{attribute addProperty BoxType "EK1122-0000-0018"}
{attribute addProperty Id "A_0155_AX5191_0000_0212_AX5191_0000_0212AX5191_3FB01CDA28235.25Beckhoff_AX5xxxsub_EK1100EK1100_179A0949162A_0154_AX5118_0000_0011AX5118_47F5CC4725031.25A_0155_AX5125_0000_0011AX5125_47F5CC4725031.25A_0156_AX5201_0000_0011AX5201_D0280DF235444.25A_0157_AX5106_0000_0010AX5106_47F5CC4725031.25A_0158_AX5112_0000_0010AX5112_47F5CC4725031.25A_0159_AX5118_0000_0010AX5118_47F5CC4725031.25A_0160_AX5112_0000_0008AX5112_47F5CC4725031.25A_0161_AX5103_0000_0007AX5103_47F5CC4725031.25A_0162_AX5118_0000_0007AX5118_47F5CC4725031.25A_0163_AX5106_0000_0006AX5106_47F5CC4725031.25A_0164_AX5112_0000_0006AX5112_47F5CC4725031.25A_0165_AX5201_0000_0006AX5201_D0280DF235444.25A_0166_AX5101_0000_0005AX5101_47F5CC4725031.25A_0167_AX5103_0000_0005AX5103_47F5CC4725031.25A_0168_AX5203_0000_0005AX5203_D0280DF235444.25A_0169_AX5206_0000_0005AX5206_D0280DF235444.25A_0170_AX5101_0000_0004AX5101_47F5CC4725031.25A_0171_AX5103_0000_0004AX5103_47F5CC4725031.25A_0172_AX5206_0000_0004AX5206_D0280DF235444.25A_0173_AX5101_0000_0003AX5101_47F5CC4725031.25A_0174_AX5103_0000_0003AX5103_47F5CC4725031.25A_0175_AX5201_0000_0003AX5201_D0280DF235444.25A_0176_AX5203_0000_0003AX5203_D0280DF235444.25A_0177_AX5021_0000_0002AX5021_292ACD4718623.25A_0153_AX5206_0000_0200AX5206_7BA2318041852.25A_0152_AX5140_0000_0200AX5140_3FB01CDA28235.25A_0151_AX5118_0000_0200AX5118_3FB01CDA28235.25A_0150_AX5125_0000_0201AX5125_3FB01CDA28235.25A_0149_AX5101_0000_0202AX5101_3FB01CDA28235.25A_0148_AX5206_0000_0203AX5206_7BA2318041852.25A_0147_AX5172_0000_0203AX5172_3FB01CDA28235.25A_0146_AX5106_0000_0203AX5106_3FB01CDA28235.25A_0145_AX5206_0000_0210AX5206_7BA2318041852.25A_0144_AX5203_0000_0210AX5203_7BA2318041852.25A_0143_AX5193_0000_0210AX5193_3FB01CDA28235.25A_0142_AX5192_0000_0210AX5192_3FB01CDA28235.25A_0141_AX5191_0000_0210AX5191_3FB01CDA28235.25A_0140_AX5160_0000_0210AX5160_3FB01CDA28235.25A_0139_AX5140_0000_0210AX5140_3FB01CDA28235.25A_0138_AX5125_0000_0210AX5125_3FB01CDA28235.25A_0137_AX5112_0000_0210AX5112_3FB01CDA28235.25A_0136_AX5101_0000_0210AX5101_3FB01CDA28235.25A_0135_AX5206_0000_0212AX5206_7BA2318041852.25A_0134_AX5203_0000_0212AX5203_7BA2318041852.25A_0133_AX5172_0000_0212AX5172_3FB01CDA28235.25A_0132_AX5160_0000_0212AX5160_3FB01CDA28235.25A_0131_AX5125_0000_0212AX5125_3FB01CDA28235.25A_0130_AX5118_0000_0212AX5118_3FB01CDA28235.25A_0129_AX5106_0000_0212AX5106_3FB01CDA28235.25A_0128_AX5206_0000_0213AX5206_7BA2318041852.25A_0127_AX5101_0000_0213AX5101_3FB01CDA28235.25A_0081_AX5101_0000_0012AX5101_47F5CC4725031.25A_0082_AX5103_0000_0012AX5103_47F5CC4725031.25A_0083_AX5203_0000_0012AX5203_D0280DF235444.25A_0084_AX5101_0000_0011AX5101_47F5CC4725031.25A_0085_AX5203_0000_0011AX5203_D0280DF235444.25A_0086_AX5206_0000_0011AX5206_D0280DF235444.25A_0087_AX5101_0000_0010AX5101_47F5CC4725031.25A_0088_AX5103_0000_0010AX5103_47F5CC4725031.25A_0089_AX5125_0000_0010AX5125_47F5CC4725031.25A_0090_AX5201_0000_0010AX5201_D0280DF235444.25A_0091_AX5203_0000_0010AX5203_D0280DF235444.25A_0092_AX5206_0000_0010AX5206_D0280DF235444.25A_0093_AX5101_0000_0009AX5101_47F5CC4725031.25A_0094_AX5103_0000_0009AX5103_47F5CC4725031.25A_0095_AX5106_0000_0009AX5106_47F5CC4725031.25A_0096_AX5112_0000_0009AX5112_47F5CC4725031.25A_0097_AX5118_0000_0009AX5118_47F5CC4725031.25A_0098_AX5125_0000_0009AX5125_47F5CC4725031.25A_0099_AX5201_0000_0009AX5201_D0280DF235444.25A_0100_AX5203_0000_0009AX5203_D0280DF235444.25A_0101_AX5206_0000_0009AX5206_D0280DF235444.25A_0102_AX5101_0000_0008AX5101_47F5CC4725031.25A_0103_AX5103_0000_0008AX5103_47F5CC4725031.25A_0104_AX5106_0000_0008AX5106_47F5CC4725031.25A_0105_AX5118_0000_0008AX5118_47F5CC4725031.25A_0106_AX5125_0000_0008AX5125_47F5CC4725031.25A_0107_AX5201_0000_0008AX5201_D0280DF235444.25A_0108_AX5203_0000_0008AX5203_D0280DF235444.25A_0109_AX5206_0000_0008AX5206_D0280DF235444.25A_0110_AX5101_0000_0007AX5101_47F5CC4725031.25A_0111_AX5106_0000_0007AX5106_47F5CC4725031.25A_0112_AX5112_0000_0007AX5112_47F5CC4725031.25A_0113_AX5125_0000_0007AX5125_47F5CC4725031.25A_0114_AX5201_0000_0007AX5201_D0280DF235444.25A_0115_AX5203_0000_0007AX5203_D0280DF235444.25A_0116_AX5206_0000_0007AX5206_D0280DF235444.25A_0117_AX5101_0000_0006AX5101_47F5CC4725031.25A_0118_AX5103_0000_0006AX5103_47F5CC4725031.25A_0119_AX5203_0000_0006AX5203_D0280DF235444.25A_0120_AX5206_0000_0006AX5206_D0280DF235444.25A_0121_AX5106_0000_0005AX5106_47F5CC4725031.25A_0122_AX5201_0000_0005AX5201_D0280DF235444.25A_0123_AX5106_0000_0004AX5106_47F5CC4725031.25A_0124_AX5201_0000_0004AX5201_D0280DF235444.25A_0125_AX5203_0000_0004AX5203_D0280DF235444.25A_0126_AX5021_0000_0001AX5021_292ACD4718623.25A_0080_AX5203_0000_0200AX5203_7BA2318041852.25A_0079_AX5201_0000_0200AX5201_7BA2318041852.25A_0078_AX5125_0000_0200AX5125_3FB01CDA28235.25A_0077_AX5106_0000_0200AX5106_3FB01CDA28235.25A_0076_AX5101_0000_0200AX5101_3FB01CDA28235.25A_0075_AX5206_0000_0201AX5206_7BA2318041852.25A_0074_AX5203_0000_0201AX5203_7BA2318041852.25A_0073_AX5201_0000_0201AX5201_7BA2318041852.25A_0072_AX5172_0000_0201AX5172_3FB01CDA28235.25A_0071_AX5160_0000_0201AX5160_3FB01CDA28235.25A_0070_AX5140_0000_0201AX5140_3FB01CDA28235.25A_0069_AX5112_0000_0201AX5112_3FB01CDA28235.25A_0068_AX5103_0000_0201AX5103_3FB01CDA28235.25A_0067_AX5101_0000_0201AX5101_3FB01CDA28235.25A_0066_AX5206_0000_0202AX5206_7BA2318041852.25A_0065_AX5203_0000_0202AX5203_7BA2318041852.25A_0064_AX5201_0000_0202AX5201_7BA2318041852.25A_0063_AX5172_0000_0202AX5172_3FB01CDA28235.25A_0062_AX5160_0000_0202AX5160_3FB01CDA28235.25A_0061_AX5140_0000_0202AX5140_3FB01CDA28235.25A_0060_AX5125_0000_0202AX5125_3FB01CDA28235.25A_0059_AX5118_0000_0202AX5118_3FB01CDA28235.25A_0058_AX5112_0000_0202AX5112_3FB01CDA28235.25A_0057_AX5106_0000_0202AX5106_3FB01CDA28235.25A_0056_AX5103_0000_0202AX5103_3FB01CDA28235.25A_0055_AX5203_0000_0203AX5203_7BA2318041852.25A_0054_AX5201_0000_0203AX5201_7BA2318041852.25A_0053_AX5192_0000_0203AX5192_3FB01CDA28235.25A_0052_AX5191_0000_0203AX5191_3FB01CDA28235.25A_0051_AX5190_0000_0203AX5190_3FB01CDA28235.25A_0050_AX5160_0000_0203AX5160_3FB01CDA28235.25A_0049_AX5140_0000_0203AX5140_3FB01CDA28235.25A_0048_AX5125_0000_0203AX5125_3FB01CDA28235.25A_0047_AX5118_0000_0203AX5118_3FB01CDA28235.25A_0046_AX5112_0000_0203AX5112_3FB01CDA28235.25A_0045_AX5103_0000_0203AX5103_3FB01CDA28235.25A_0044_AX5101_0000_0203AX5101_3FB01CDA28235.25A_0043_AX5201_0000_0210AX5201_7BA2318041852.25A_0042_AX5190_0000_0210AX5190_3FB01CDA28235.25A_0041_AX5172_0000_0210AX5172_3FB01CDA28235.25A_0040_AX5118_0000_0210AX5118_3FB01CDA28235.25A_0039_AX5106_0000_0210AX5106_3FB01CDA28235.25A_0038_AX5201_0000_0212AX5201_7BA2318041852.25A_0037_AX5193_0000_0212AX5193_3FB01CDA28235.25A_0036_AX5192_0000_0212AX5192_3FB01CDA28235.25A_0035_AX5190_0000_0212AX5190_3FB01CDA28235.25A_0034_AX5140_0000_0212AX5140_3FB01CDA28235.25A_0033_AX5112_0000_0212AX5112_3FB01CDA28235.25A_0032_AX5103_0000_0212AX5103_3FB01CDA28235.25A_0031_AX5101_0000_0212AX5101_3FB01CDA28235.25A_0030_AX5203_0000_0213AX5203_7BA2318041852.25A_0029_AX5201_0000_0213AX5201_7BA2318041852.25A_0028_AX5193_0000_0213AX5193_3FB01CDA28235.25A_0027_AX5192_0000_0213AX5192_3FB01CDA28235.25A_0026_AX5191_0000_0213AX5191_3FB01CDA28235.25A_0025_AX5190_0000_0213AX5190_3FB01CDA28235.25A_0024_AX5172_0000_0213AX5172_3FB01CDA28235.25A_0023_AX5160_0000_0213AX5160_3FB01CDA28235.25A_0022_AX5140_0000_0213AX5140_3FB01CDA28235.25A_0021_AX5125_0000_0213AX5125_3FB01CDA28235.25A_0020_AX5118_0000_0213AX5118_3FB01CDA28235.25A_0019_AX5112_0000_0213AX5112_3FB01CDA28235.25A_0018_AX5106_0000_0213AX5106_3FB01CDA28235.25A_0017_AX5103_0000_0213AX5103_3FB01CDA28235.25A_0016_AX5206_0000_0214AX5206_7BA2318041852.25A_0015_AX5203_0000_0214AX5203_7BA2318041852.25A_0014_AX5201_0000_0214AX5201_7BA2318041852.25A_0013_AX5193_0000_0214AX5193_3FB01CDA28235.25A_0012_AX5192_0000_0214AX5192_3FB01CDA28235.25A_0011_AX5191_0000_0214AX5191_3FB01CDA28235.25A_0010_AX5190_0000_0214AX5190_3FB01CDA28235.25A_0009_AX5172_0000_0214AX5172_3FB01CDA28235.25A_0008_AX5160_0000_0214AX5160_3FB01CDA28235.25A_0007_AX5140_0000_0214AX5140_3FB01CDA28235.25A_0006_AX5125_0000_0214AX5125_3FB01CDA28235.25A_0005_AX5118_0000_0214AX5118_3FB01CDA28235.25A_0004_AX5112_0000_0214AX5112_3FB01CDA28235.25A_0003_AX5106_0000_0214AX5106_3FB01CDA28235.25A_0002_AX5103_0000_0214AX5103_3FB01CDA28235.25A_0001_AX5101_0000_0214AX5101_3FB01CDA28235.25A_0156_AX5103_0000_0210_AX5103_0000_0210AX5103_3FB01CDA28235.25A_0157_AX5193_0000_0203_AX5193_0000_0203AX5193_3FB01CDA28235.25A_0158_AX5106_0000_0201_AX5106_0000_0201AX5106_3FB01CDA28235.25A_0159_AX5118_0000_0201_AX5118_0000_0201AX5118_3FB01CDA28235.25A_0160_AX5103_0000_0200_AX5103_0000_0200AX5103_3FB01CDA28235.25A_0161_AX5112_0000_0200_AX5112_0000_0200AX5112_3FB01CDA28235.25A_0162_AX5106_0000_0012_AX5106_0000_0012AX5106_47F5CC4725031.25A_0163_AX5112_0000_0012_AX5112_0000_0012AX5112_47F5CC4725031.25A_0164_AX5118_0000_0012_AX5118_0000_0012AX5118_47F5CC4725031.25A_0165_AX5125_0000_0012_AX5125_0000_0012AX5125_47F5CC4725031.25A_0166_AX5201_0000_0012_AX5201_0000_0012AX5201_D0280DF235444.25A_0167_AX5206_0000_0012_AX5206_0000_0012AX5206_D0280DF235444.25A_0168_AX5103_0000_0011AX5103_47F5CC4725031.25A_0169_AX5106_0000_0011_AX5106_0000_0011AX5106_47F5CC4725031.25A_0170_AX5112_0000_0011_AX5112_0000_0011AX5112_47F5CC4725031.25A_0171_AX5106_0000_0003_AX5106_0000_0003AX5106_47F5CC4725031.25A_0172_AX5206_0000_0003_AX5206_0000_0003AX5206_D0280DF235444.25"}
{attribute addProperty CRC "1593486659"}
{attribute addProperty SizeInBites "58670"}
{attribute addProperty SizeInBytes "7333.75"}
TYPE Beckhoff_AX5xxxEK1122_5EFAAD43 EXTENDS EK1122_179A0949 :
STRUCT
	{attribute addProperty Name "A_0155_AX5191_0000_0212_AX5191_0000_0212"}
	A_0155_AX5191_0000_0212_AX5191_0000_0212 : AX5191_3FB01CDA;
	{attribute addProperty Name "Beckhoff_AX5xxxsub_EK1100"}
	Beckhoff_AX5xxxsub_EK1100 : EK1100_179A0949;
	{attribute addProperty Name "A_0154_AX5118_0000_0011"}
	A_0154_AX5118_0000_0011 : AX5118_47F5CC47;
	{attribute addProperty Name "A_0155_AX5125_0000_0011"}
	A_0155_AX5125_0000_0011 : AX5125_47F5CC47;
	{attribute addProperty Name "A_0156_AX5201_0000_0011"}
	A_0156_AX5201_0000_0011 : AX5201_D0280DF2;
	{attribute addProperty Name "A_0157_AX5106_0000_0010"}
	A_0157_AX5106_0000_0010 : AX5106_47F5CC47;
	{attribute addProperty Name "A_0158_AX5112_0000_0010"}
	A_0158_AX5112_0000_0010 : AX5112_47F5CC47;
	{attribute addProperty Name "A_0159_AX5118_0000_0010"}
	A_0159_AX5118_0000_0010 : AX5118_47F5CC47;
	{attribute addProperty Name "A_0160_AX5112_0000_0008"}
	A_0160_AX5112_0000_0008 : AX5112_47F5CC47;
	{attribute addProperty Name "A_0161_AX5103_0000_0007"}
	A_0161_AX5103_0000_0007 : AX5103_47F5CC47;
	{attribute addProperty Name "A_0162_AX5118_0000_0007"}
	A_0162_AX5118_0000_0007 : AX5118_47F5CC47;
	{attribute addProperty Name "A_0163_AX5106_0000_0006"}
	A_0163_AX5106_0000_0006 : AX5106_47F5CC47;
	{attribute addProperty Name "A_0164_AX5112_0000_0006"}
	A_0164_AX5112_0000_0006 : AX5112_47F5CC47;
	{attribute addProperty Name "A_0165_AX5201_0000_0006"}
	A_0165_AX5201_0000_0006 : AX5201_D0280DF2;
	{attribute addProperty Name "A_0166_AX5101_0000_0005"}
	A_0166_AX5101_0000_0005 : AX5101_47F5CC47;
	{attribute addProperty Name "A_0167_AX5103_0000_0005"}
	A_0167_AX5103_0000_0005 : AX5103_47F5CC47;
	{attribute addProperty Name "A_0168_AX5203_0000_0005"}
	A_0168_AX5203_0000_0005 : AX5203_D0280DF2;
	{attribute addProperty Name "A_0169_AX5206_0000_0005"}
	A_0169_AX5206_0000_0005 : AX5206_D0280DF2;
	{attribute addProperty Name "A_0170_AX5101_0000_0004"}
	A_0170_AX5101_0000_0004 : AX5101_47F5CC47;
	{attribute addProperty Name "A_0171_AX5103_0000_0004"}
	A_0171_AX5103_0000_0004 : AX5103_47F5CC47;
	{attribute addProperty Name "A_0172_AX5206_0000_0004"}
	A_0172_AX5206_0000_0004 : AX5206_D0280DF2;
	{attribute addProperty Name "A_0173_AX5101_0000_0003"}
	A_0173_AX5101_0000_0003 : AX5101_47F5CC47;
	{attribute addProperty Name "A_0174_AX5103_0000_0003"}
	A_0174_AX5103_0000_0003 : AX5103_47F5CC47;
	{attribute addProperty Name "A_0175_AX5201_0000_0003"}
	A_0175_AX5201_0000_0003 : AX5201_D0280DF2;
	{attribute addProperty Name "A_0176_AX5203_0000_0003"}
	A_0176_AX5203_0000_0003 : AX5203_D0280DF2;
	{attribute addProperty Name "A_0177_AX5021_0000_0002"}
	A_0177_AX5021_0000_0002 : AX5021_292ACD47;
	{attribute addProperty Name "A_0153_AX5206_0000_0200"}
	A_0153_AX5206_0000_0200 : AX5206_7BA23180;
	{attribute addProperty Name "A_0152_AX5140_0000_0200"}
	A_0152_AX5140_0000_0200 : AX5140_3FB01CDA;
	{attribute addProperty Name "A_0151_AX5118_0000_0200"}
	A_0151_AX5118_0000_0200 : AX5118_3FB01CDA;
	{attribute addProperty Name "A_0150_AX5125_0000_0201"}
	A_0150_AX5125_0000_0201 : AX5125_3FB01CDA;
	{attribute addProperty Name "A_0149_AX5101_0000_0202"}
	A_0149_AX5101_0000_0202 : AX5101_3FB01CDA;
	{attribute addProperty Name "A_0148_AX5206_0000_0203"}
	A_0148_AX5206_0000_0203 : AX5206_7BA23180;
	{attribute addProperty Name "A_0147_AX5172_0000_0203"}
	A_0147_AX5172_0000_0203 : AX5172_3FB01CDA;
	{attribute addProperty Name "A_0146_AX5106_0000_0203"}
	A_0146_AX5106_0000_0203 : AX5106_3FB01CDA;
	{attribute addProperty Name "A_0145_AX5206_0000_0210"}
	A_0145_AX5206_0000_0210 : AX5206_7BA23180;
	{attribute addProperty Name "A_0144_AX5203_0000_0210"}
	A_0144_AX5203_0000_0210 : AX5203_7BA23180;
	{attribute addProperty Name "A_0143_AX5193_0000_0210"}
	A_0143_AX5193_0000_0210 : AX5193_3FB01CDA;
	{attribute addProperty Name "A_0142_AX5192_0000_0210"}
	A_0142_AX5192_0000_0210 : AX5192_3FB01CDA;
	{attribute addProperty Name "A_0141_AX5191_0000_0210"}
	A_0141_AX5191_0000_0210 : AX5191_3FB01CDA;
	{attribute addProperty Name "A_0140_AX5160_0000_0210"}
	A_0140_AX5160_0000_0210 : AX5160_3FB01CDA;
	{attribute addProperty Name "A_0139_AX5140_0000_0210"}
	A_0139_AX5140_0000_0210 : AX5140_3FB01CDA;
	{attribute addProperty Name "A_0138_AX5125_0000_0210"}
	A_0138_AX5125_0000_0210 : AX5125_3FB01CDA;
	{attribute addProperty Name "A_0137_AX5112_0000_0210"}
	A_0137_AX5112_0000_0210 : AX5112_3FB01CDA;
	{attribute addProperty Name "A_0136_AX5101_0000_0210"}
	A_0136_AX5101_0000_0210 : AX5101_3FB01CDA;
	{attribute addProperty Name "A_0135_AX5206_0000_0212"}
	A_0135_AX5206_0000_0212 : AX5206_7BA23180;
	{attribute addProperty Name "A_0134_AX5203_0000_0212"}
	A_0134_AX5203_0000_0212 : AX5203_7BA23180;
	{attribute addProperty Name "A_0133_AX5172_0000_0212"}
	A_0133_AX5172_0000_0212 : AX5172_3FB01CDA;
	{attribute addProperty Name "A_0132_AX5160_0000_0212"}
	A_0132_AX5160_0000_0212 : AX5160_3FB01CDA;
	{attribute addProperty Name "A_0131_AX5125_0000_0212"}
	A_0131_AX5125_0000_0212 : AX5125_3FB01CDA;
	{attribute addProperty Name "A_0130_AX5118_0000_0212"}
	A_0130_AX5118_0000_0212 : AX5118_3FB01CDA;
	{attribute addProperty Name "A_0129_AX5106_0000_0212"}
	A_0129_AX5106_0000_0212 : AX5106_3FB01CDA;
	{attribute addProperty Name "A_0128_AX5206_0000_0213"}
	A_0128_AX5206_0000_0213 : AX5206_7BA23180;
	{attribute addProperty Name "A_0127_AX5101_0000_0213"}
	A_0127_AX5101_0000_0213 : AX5101_3FB01CDA;
	{attribute addProperty Name "A_0081_AX5101_0000_0012"}
	A_0081_AX5101_0000_0012 : AX5101_47F5CC47;
	{attribute addProperty Name "A_0082_AX5103_0000_0012"}
	A_0082_AX5103_0000_0012 : AX5103_47F5CC47;
	{attribute addProperty Name "A_0083_AX5203_0000_0012"}
	A_0083_AX5203_0000_0012 : AX5203_D0280DF2;
	{attribute addProperty Name "A_0084_AX5101_0000_0011"}
	A_0084_AX5101_0000_0011 : AX5101_47F5CC47;
	{attribute addProperty Name "A_0085_AX5203_0000_0011"}
	A_0085_AX5203_0000_0011 : AX5203_D0280DF2;
	{attribute addProperty Name "A_0086_AX5206_0000_0011"}
	A_0086_AX5206_0000_0011 : AX5206_D0280DF2;
	{attribute addProperty Name "A_0087_AX5101_0000_0010"}
	A_0087_AX5101_0000_0010 : AX5101_47F5CC47;
	{attribute addProperty Name "A_0088_AX5103_0000_0010"}
	A_0088_AX5103_0000_0010 : AX5103_47F5CC47;
	{attribute addProperty Name "A_0089_AX5125_0000_0010"}
	A_0089_AX5125_0000_0010 : AX5125_47F5CC47;
	{attribute addProperty Name "A_0090_AX5201_0000_0010"}
	A_0090_AX5201_0000_0010 : AX5201_D0280DF2;
	{attribute addProperty Name "A_0091_AX5203_0000_0010"}
	A_0091_AX5203_0000_0010 : AX5203_D0280DF2;
	{attribute addProperty Name "A_0092_AX5206_0000_0010"}
	A_0092_AX5206_0000_0010 : AX5206_D0280DF2;
	{attribute addProperty Name "A_0093_AX5101_0000_0009"}
	A_0093_AX5101_0000_0009 : AX5101_47F5CC47;
	{attribute addProperty Name "A_0094_AX5103_0000_0009"}
	A_0094_AX5103_0000_0009 : AX5103_47F5CC47;
	{attribute addProperty Name "A_0095_AX5106_0000_0009"}
	A_0095_AX5106_0000_0009 : AX5106_47F5CC47;
	{attribute addProperty Name "A_0096_AX5112_0000_0009"}
	A_0096_AX5112_0000_0009 : AX5112_47F5CC47;
	{attribute addProperty Name "A_0097_AX5118_0000_0009"}
	A_0097_AX5118_0000_0009 : AX5118_47F5CC47;
	{attribute addProperty Name "A_0098_AX5125_0000_0009"}
	A_0098_AX5125_0000_0009 : AX5125_47F5CC47;
	{attribute addProperty Name "A_0099_AX5201_0000_0009"}
	A_0099_AX5201_0000_0009 : AX5201_D0280DF2;
	{attribute addProperty Name "A_0100_AX5203_0000_0009"}
	A_0100_AX5203_0000_0009 : AX5203_D0280DF2;
	{attribute addProperty Name "A_0101_AX5206_0000_0009"}
	A_0101_AX5206_0000_0009 : AX5206_D0280DF2;
	{attribute addProperty Name "A_0102_AX5101_0000_0008"}
	A_0102_AX5101_0000_0008 : AX5101_47F5CC47;
	{attribute addProperty Name "A_0103_AX5103_0000_0008"}
	A_0103_AX5103_0000_0008 : AX5103_47F5CC47;
	{attribute addProperty Name "A_0104_AX5106_0000_0008"}
	A_0104_AX5106_0000_0008 : AX5106_47F5CC47;
	{attribute addProperty Name "A_0105_AX5118_0000_0008"}
	A_0105_AX5118_0000_0008 : AX5118_47F5CC47;
	{attribute addProperty Name "A_0106_AX5125_0000_0008"}
	A_0106_AX5125_0000_0008 : AX5125_47F5CC47;
	{attribute addProperty Name "A_0107_AX5201_0000_0008"}
	A_0107_AX5201_0000_0008 : AX5201_D0280DF2;
	{attribute addProperty Name "A_0108_AX5203_0000_0008"}
	A_0108_AX5203_0000_0008 : AX5203_D0280DF2;
	{attribute addProperty Name "A_0109_AX5206_0000_0008"}
	A_0109_AX5206_0000_0008 : AX5206_D0280DF2;
	{attribute addProperty Name "A_0110_AX5101_0000_0007"}
	A_0110_AX5101_0000_0007 : AX5101_47F5CC47;
	{attribute addProperty Name "A_0111_AX5106_0000_0007"}
	A_0111_AX5106_0000_0007 : AX5106_47F5CC47;
	{attribute addProperty Name "A_0112_AX5112_0000_0007"}
	A_0112_AX5112_0000_0007 : AX5112_47F5CC47;
	{attribute addProperty Name "A_0113_AX5125_0000_0007"}
	A_0113_AX5125_0000_0007 : AX5125_47F5CC47;
	{attribute addProperty Name "A_0114_AX5201_0000_0007"}
	A_0114_AX5201_0000_0007 : AX5201_D0280DF2;
	{attribute addProperty Name "A_0115_AX5203_0000_0007"}
	A_0115_AX5203_0000_0007 : AX5203_D0280DF2;
	{attribute addProperty Name "A_0116_AX5206_0000_0007"}
	A_0116_AX5206_0000_0007 : AX5206_D0280DF2;
	{attribute addProperty Name "A_0117_AX5101_0000_0006"}
	A_0117_AX5101_0000_0006 : AX5101_47F5CC47;
	{attribute addProperty Name "A_0118_AX5103_0000_0006"}
	A_0118_AX5103_0000_0006 : AX5103_47F5CC47;
	{attribute addProperty Name "A_0119_AX5203_0000_0006"}
	A_0119_AX5203_0000_0006 : AX5203_D0280DF2;
	{attribute addProperty Name "A_0120_AX5206_0000_0006"}
	A_0120_AX5206_0000_0006 : AX5206_D0280DF2;
	{attribute addProperty Name "A_0121_AX5106_0000_0005"}
	A_0121_AX5106_0000_0005 : AX5106_47F5CC47;
	{attribute addProperty Name "A_0122_AX5201_0000_0005"}
	A_0122_AX5201_0000_0005 : AX5201_D0280DF2;
	{attribute addProperty Name "A_0123_AX5106_0000_0004"}
	A_0123_AX5106_0000_0004 : AX5106_47F5CC47;
	{attribute addProperty Name "A_0124_AX5201_0000_0004"}
	A_0124_AX5201_0000_0004 : AX5201_D0280DF2;
	{attribute addProperty Name "A_0125_AX5203_0000_0004"}
	A_0125_AX5203_0000_0004 : AX5203_D0280DF2;
	{attribute addProperty Name "A_0126_AX5021_0000_0001"}
	A_0126_AX5021_0000_0001 : AX5021_292ACD47;
	{attribute addProperty Name "A_0080_AX5203_0000_0200"}
	A_0080_AX5203_0000_0200 : AX5203_7BA23180;
	{attribute addProperty Name "A_0079_AX5201_0000_0200"}
	A_0079_AX5201_0000_0200 : AX5201_7BA23180;
	{attribute addProperty Name "A_0078_AX5125_0000_0200"}
	A_0078_AX5125_0000_0200 : AX5125_3FB01CDA;
	{attribute addProperty Name "A_0077_AX5106_0000_0200"}
	A_0077_AX5106_0000_0200 : AX5106_3FB01CDA;
	{attribute addProperty Name "A_0076_AX5101_0000_0200"}
	A_0076_AX5101_0000_0200 : AX5101_3FB01CDA;
	{attribute addProperty Name "A_0075_AX5206_0000_0201"}
	A_0075_AX5206_0000_0201 : AX5206_7BA23180;
	{attribute addProperty Name "A_0074_AX5203_0000_0201"}
	A_0074_AX5203_0000_0201 : AX5203_7BA23180;
	{attribute addProperty Name "A_0073_AX5201_0000_0201"}
	A_0073_AX5201_0000_0201 : AX5201_7BA23180;
	{attribute addProperty Name "A_0072_AX5172_0000_0201"}
	A_0072_AX5172_0000_0201 : AX5172_3FB01CDA;
	{attribute addProperty Name "A_0071_AX5160_0000_0201"}
	A_0071_AX5160_0000_0201 : AX5160_3FB01CDA;
	{attribute addProperty Name "A_0070_AX5140_0000_0201"}
	A_0070_AX5140_0000_0201 : AX5140_3FB01CDA;
	{attribute addProperty Name "A_0069_AX5112_0000_0201"}
	A_0069_AX5112_0000_0201 : AX5112_3FB01CDA;
	{attribute addProperty Name "A_0068_AX5103_0000_0201"}
	A_0068_AX5103_0000_0201 : AX5103_3FB01CDA;
	{attribute addProperty Name "A_0067_AX5101_0000_0201"}
	A_0067_AX5101_0000_0201 : AX5101_3FB01CDA;
	{attribute addProperty Name "A_0066_AX5206_0000_0202"}
	A_0066_AX5206_0000_0202 : AX5206_7BA23180;
	{attribute addProperty Name "A_0065_AX5203_0000_0202"}
	A_0065_AX5203_0000_0202 : AX5203_7BA23180;
	{attribute addProperty Name "A_0064_AX5201_0000_0202"}
	A_0064_AX5201_0000_0202 : AX5201_7BA23180;
	{attribute addProperty Name "A_0063_AX5172_0000_0202"}
	A_0063_AX5172_0000_0202 : AX5172_3FB01CDA;
	{attribute addProperty Name "A_0062_AX5160_0000_0202"}
	A_0062_AX5160_0000_0202 : AX5160_3FB01CDA;
	{attribute addProperty Name "A_0061_AX5140_0000_0202"}
	A_0061_AX5140_0000_0202 : AX5140_3FB01CDA;
	{attribute addProperty Name "A_0060_AX5125_0000_0202"}
	A_0060_AX5125_0000_0202 : AX5125_3FB01CDA;
	{attribute addProperty Name "A_0059_AX5118_0000_0202"}
	A_0059_AX5118_0000_0202 : AX5118_3FB01CDA;
	{attribute addProperty Name "A_0058_AX5112_0000_0202"}
	A_0058_AX5112_0000_0202 : AX5112_3FB01CDA;
	{attribute addProperty Name "A_0057_AX5106_0000_0202"}
	A_0057_AX5106_0000_0202 : AX5106_3FB01CDA;
	{attribute addProperty Name "A_0056_AX5103_0000_0202"}
	A_0056_AX5103_0000_0202 : AX5103_3FB01CDA;
	{attribute addProperty Name "A_0055_AX5203_0000_0203"}
	A_0055_AX5203_0000_0203 : AX5203_7BA23180;
	{attribute addProperty Name "A_0054_AX5201_0000_0203"}
	A_0054_AX5201_0000_0203 : AX5201_7BA23180;
	{attribute addProperty Name "A_0053_AX5192_0000_0203"}
	A_0053_AX5192_0000_0203 : AX5192_3FB01CDA;
	{attribute addProperty Name "A_0052_AX5191_0000_0203"}
	A_0052_AX5191_0000_0203 : AX5191_3FB01CDA;
	{attribute addProperty Name "A_0051_AX5190_0000_0203"}
	A_0051_AX5190_0000_0203 : AX5190_3FB01CDA;
	{attribute addProperty Name "A_0050_AX5160_0000_0203"}
	A_0050_AX5160_0000_0203 : AX5160_3FB01CDA;
	{attribute addProperty Name "A_0049_AX5140_0000_0203"}
	A_0049_AX5140_0000_0203 : AX5140_3FB01CDA;
	{attribute addProperty Name "A_0048_AX5125_0000_0203"}
	A_0048_AX5125_0000_0203 : AX5125_3FB01CDA;
	{attribute addProperty Name "A_0047_AX5118_0000_0203"}
	A_0047_AX5118_0000_0203 : AX5118_3FB01CDA;
	{attribute addProperty Name "A_0046_AX5112_0000_0203"}
	A_0046_AX5112_0000_0203 : AX5112_3FB01CDA;
	{attribute addProperty Name "A_0045_AX5103_0000_0203"}
	A_0045_AX5103_0000_0203 : AX5103_3FB01CDA;
	{attribute addProperty Name "A_0044_AX5101_0000_0203"}
	A_0044_AX5101_0000_0203 : AX5101_3FB01CDA;
	{attribute addProperty Name "A_0043_AX5201_0000_0210"}
	A_0043_AX5201_0000_0210 : AX5201_7BA23180;
	{attribute addProperty Name "A_0042_AX5190_0000_0210"}
	A_0042_AX5190_0000_0210 : AX5190_3FB01CDA;
	{attribute addProperty Name "A_0041_AX5172_0000_0210"}
	A_0041_AX5172_0000_0210 : AX5172_3FB01CDA;
	{attribute addProperty Name "A_0040_AX5118_0000_0210"}
	A_0040_AX5118_0000_0210 : AX5118_3FB01CDA;
	{attribute addProperty Name "A_0039_AX5106_0000_0210"}
	A_0039_AX5106_0000_0210 : AX5106_3FB01CDA;
	{attribute addProperty Name "A_0038_AX5201_0000_0212"}
	A_0038_AX5201_0000_0212 : AX5201_7BA23180;
	{attribute addProperty Name "A_0037_AX5193_0000_0212"}
	A_0037_AX5193_0000_0212 : AX5193_3FB01CDA;
	{attribute addProperty Name "A_0036_AX5192_0000_0212"}
	A_0036_AX5192_0000_0212 : AX5192_3FB01CDA;
	{attribute addProperty Name "A_0035_AX5190_0000_0212"}
	A_0035_AX5190_0000_0212 : AX5190_3FB01CDA;
	{attribute addProperty Name "A_0034_AX5140_0000_0212"}
	A_0034_AX5140_0000_0212 : AX5140_3FB01CDA;
	{attribute addProperty Name "A_0033_AX5112_0000_0212"}
	A_0033_AX5112_0000_0212 : AX5112_3FB01CDA;
	{attribute addProperty Name "A_0032_AX5103_0000_0212"}
	A_0032_AX5103_0000_0212 : AX5103_3FB01CDA;
	{attribute addProperty Name "A_0031_AX5101_0000_0212"}
	A_0031_AX5101_0000_0212 : AX5101_3FB01CDA;
	{attribute addProperty Name "A_0030_AX5203_0000_0213"}
	A_0030_AX5203_0000_0213 : AX5203_7BA23180;
	{attribute addProperty Name "A_0029_AX5201_0000_0213"}
	A_0029_AX5201_0000_0213 : AX5201_7BA23180;
	{attribute addProperty Name "A_0028_AX5193_0000_0213"}
	A_0028_AX5193_0000_0213 : AX5193_3FB01CDA;
	{attribute addProperty Name "A_0027_AX5192_0000_0213"}
	A_0027_AX5192_0000_0213 : AX5192_3FB01CDA;
	{attribute addProperty Name "A_0026_AX5191_0000_0213"}
	A_0026_AX5191_0000_0213 : AX5191_3FB01CDA;
	{attribute addProperty Name "A_0025_AX5190_0000_0213"}
	A_0025_AX5190_0000_0213 : AX5190_3FB01CDA;
	{attribute addProperty Name "A_0024_AX5172_0000_0213"}
	A_0024_AX5172_0000_0213 : AX5172_3FB01CDA;
	{attribute addProperty Name "A_0023_AX5160_0000_0213"}
	A_0023_AX5160_0000_0213 : AX5160_3FB01CDA;
	{attribute addProperty Name "A_0022_AX5140_0000_0213"}
	A_0022_AX5140_0000_0213 : AX5140_3FB01CDA;
	{attribute addProperty Name "A_0021_AX5125_0000_0213"}
	A_0021_AX5125_0000_0213 : AX5125_3FB01CDA;
	{attribute addProperty Name "A_0020_AX5118_0000_0213"}
	A_0020_AX5118_0000_0213 : AX5118_3FB01CDA;
	{attribute addProperty Name "A_0019_AX5112_0000_0213"}
	A_0019_AX5112_0000_0213 : AX5112_3FB01CDA;
	{attribute addProperty Name "A_0018_AX5106_0000_0213"}
	A_0018_AX5106_0000_0213 : AX5106_3FB01CDA;
	{attribute addProperty Name "A_0017_AX5103_0000_0213"}
	A_0017_AX5103_0000_0213 : AX5103_3FB01CDA;
	{attribute addProperty Name "A_0016_AX5206_0000_0214"}
	A_0016_AX5206_0000_0214 : AX5206_7BA23180;
	{attribute addProperty Name "A_0015_AX5203_0000_0214"}
	A_0015_AX5203_0000_0214 : AX5203_7BA23180;
	{attribute addProperty Name "A_0014_AX5201_0000_0214"}
	A_0014_AX5201_0000_0214 : AX5201_7BA23180;
	{attribute addProperty Name "A_0013_AX5193_0000_0214"}
	A_0013_AX5193_0000_0214 : AX5193_3FB01CDA;
	{attribute addProperty Name "A_0012_AX5192_0000_0214"}
	A_0012_AX5192_0000_0214 : AX5192_3FB01CDA;
	{attribute addProperty Name "A_0011_AX5191_0000_0214"}
	A_0011_AX5191_0000_0214 : AX5191_3FB01CDA;
	{attribute addProperty Name "A_0010_AX5190_0000_0214"}
	A_0010_AX5190_0000_0214 : AX5190_3FB01CDA;
	{attribute addProperty Name "A_0009_AX5172_0000_0214"}
	A_0009_AX5172_0000_0214 : AX5172_3FB01CDA;
	{attribute addProperty Name "A_0008_AX5160_0000_0214"}
	A_0008_AX5160_0000_0214 : AX5160_3FB01CDA;
	{attribute addProperty Name "A_0007_AX5140_0000_0214"}
	A_0007_AX5140_0000_0214 : AX5140_3FB01CDA;
	{attribute addProperty Name "A_0006_AX5125_0000_0214"}
	A_0006_AX5125_0000_0214 : AX5125_3FB01CDA;
	{attribute addProperty Name "A_0005_AX5118_0000_0214"}
	A_0005_AX5118_0000_0214 : AX5118_3FB01CDA;
	{attribute addProperty Name "A_0004_AX5112_0000_0214"}
	A_0004_AX5112_0000_0214 : AX5112_3FB01CDA;
	{attribute addProperty Name "A_0003_AX5106_0000_0214"}
	A_0003_AX5106_0000_0214 : AX5106_3FB01CDA;
	{attribute addProperty Name "A_0002_AX5103_0000_0214"}
	A_0002_AX5103_0000_0214 : AX5103_3FB01CDA;
	{attribute addProperty Name "A_0001_AX5101_0000_0214"}
	A_0001_AX5101_0000_0214 : AX5101_3FB01CDA;
	{attribute addProperty Name "A_0156_AX5103_0000_0210_AX5103_0000_0210"}
	A_0156_AX5103_0000_0210_AX5103_0000_0210 : AX5103_3FB01CDA;
	{attribute addProperty Name "A_0157_AX5193_0000_0203_AX5193_0000_0203"}
	A_0157_AX5193_0000_0203_AX5193_0000_0203 : AX5193_3FB01CDA;
	{attribute addProperty Name "A_0158_AX5106_0000_0201_AX5106_0000_0201"}
	A_0158_AX5106_0000_0201_AX5106_0000_0201 : AX5106_3FB01CDA;
	{attribute addProperty Name "A_0159_AX5118_0000_0201_AX5118_0000_0201"}
	A_0159_AX5118_0000_0201_AX5118_0000_0201 : AX5118_3FB01CDA;
	{attribute addProperty Name "A_0160_AX5103_0000_0200_AX5103_0000_0200"}
	A_0160_AX5103_0000_0200_AX5103_0000_0200 : AX5103_3FB01CDA;
	{attribute addProperty Name "A_0161_AX5112_0000_0200_AX5112_0000_0200"}
	A_0161_AX5112_0000_0200_AX5112_0000_0200 : AX5112_3FB01CDA;
	{attribute addProperty Name "A_0162_AX5106_0000_0012_AX5106_0000_0012"}
	A_0162_AX5106_0000_0012_AX5106_0000_0012 : AX5106_47F5CC47;
	{attribute addProperty Name "A_0163_AX5112_0000_0012_AX5112_0000_0012"}
	A_0163_AX5112_0000_0012_AX5112_0000_0012 : AX5112_47F5CC47;
	{attribute addProperty Name "A_0164_AX5118_0000_0012_AX5118_0000_0012"}
	A_0164_AX5118_0000_0012_AX5118_0000_0012 : AX5118_47F5CC47;
	{attribute addProperty Name "A_0165_AX5125_0000_0012_AX5125_0000_0012"}
	A_0165_AX5125_0000_0012_AX5125_0000_0012 : AX5125_47F5CC47;
	{attribute addProperty Name "A_0166_AX5201_0000_0012_AX5201_0000_0012"}
	A_0166_AX5201_0000_0012_AX5201_0000_0012 : AX5201_D0280DF2;
	{attribute addProperty Name "A_0167_AX5206_0000_0012_AX5206_0000_0012"}
	A_0167_AX5206_0000_0012_AX5206_0000_0012 : AX5206_D0280DF2;
	{attribute addProperty Name "A_0168_AX5103_0000_0011"}
	A_0168_AX5103_0000_0011 : AX5103_47F5CC47;
	{attribute addProperty Name "A_0169_AX5106_0000_0011_AX5106_0000_0011"}
	A_0169_AX5106_0000_0011_AX5106_0000_0011 : AX5106_47F5CC47;
	{attribute addProperty Name "A_0170_AX5112_0000_0011_AX5112_0000_0011"}
	A_0170_AX5112_0000_0011_AX5112_0000_0011 : AX5112_47F5CC47;
	{attribute addProperty Name "A_0171_AX5106_0000_0003_AX5106_0000_0003"}
	A_0171_AX5106_0000_0003_AX5106_0000_0003 : AX5106_47F5CC47;
	{attribute addProperty Name "A_0172_AX5206_0000_0003_AX5206_0000_0003"}
	A_0172_AX5206_0000_0003_AX5206_0000_0003 : AX5206_D0280DF2;
END_STRUCT
END_TYPE

(* stored: Version 1.2.0.0, ProductVersion 3.1.4024.9
   DUT Beckhoff_AX5xxxEK1122_5EFAAD43: Id {e8651f54-0875-43fe-b2a9-1570eca38d40} *)
